{attribute 'linkalways'} 
{attribute 'no_explicit_call' := 'This FB is a CLASS and must be accessed using methods or properties'}
{attribute 'enable_dynamic_creation'}
FUNCTION_BLOCK _ETcVnRotationAngle EXTENDS EnumDatatypeBase
VAR
	localData : ETcVnRotationAngle;
	activeData : REFERENCE TO ETcVnRotationAngle;
	enumBaseDatatype : _DINT(localData);
END_VAR

METHOD PRIVATE AddLocalEnumeration
VAR_INPUT
	Enumeration : T_MAXSTRING;
	Value : ETcVnRotationAngle;
END_VAR
AddEnumeration(Enumeration, Value);
END_METHOD

PROPERTY PUBLIC Address : PVOID
GET
Address := ADR(activeData);
END_GET
END_PROPERTY

METHOD PUBLIC ClearReference
VAR_INPUT
END_VAR
activeData REF= localData;
SetBaseDatatypeReference();
END_METHOD

METHOD PUBLIC Clone : I_Datatype
VAR
    pClone : POINTER TO _ETcVnRotationAngle;
END_VAR
pClone := __NEW(_ETcVnRotationAngle(InitialValue := Value));
Clone := pClone^;
END_METHOD

METHOD FB_init : BOOL
VAR_INPUT
	bInitRetains : BOOL; // if TRUE, the retain variables are initialized (warm start / cold start)
	bInCopyCode : BOOL;  // if TRUE, the instance afterwards gets moved into the copy code (online change)
	InitialValue : ETcVnRotationAngle;
END_VAR
localData := InitialValue;
AddBaseDatatype(enumBaseDatatype);
ClearReference();

AddLocalEnumeration('TCVN_RA_90_DEG', ETcVnRotationAngle.TCVN_RA_90_DEG);
AddLocalEnumeration('TCVN_RA_180_DEG', ETcVnRotationAngle.TCVN_RA_180_DEG);
AddLocalEnumeration('TCVN_RA_270_DEG', ETcVnRotationAngle.TCVN_RA_270_DEG);
END_METHOD

PROPERTY PUBLIC Identifier : T_MAXSTRING
GET
Identifier := 'ETcVnRotationAngle';
END_GET
END_PROPERTY

METHOD IsEnumeratorValueEqual : BOOL
VAR_INPUT
	Enumerator : I_KeyValueForwardEnumerator;
END_VAR
VAR
	storedValue : ETcVnRotationAngle;
END_VAR
IF NOT Enumerator.TryGet(storedValue) THEN
	RETURN;
END_IF

IsEnumeratorValueEqual := storedValue = activeData;
END_METHOD

METHOD PUBLIC MakeReferenceTo
VAR_INPUT
	ReferenceTarget : REFERENCE TO ETcVnRotationAngle;
END_VAR
activeData REF= ReferenceTarget;
SetBaseDatatypeReference();
END_METHOD

METHOD PROTECTED SetBaseDatatypeReference
VAR_INPUT
END_VAR
enumBaseDatatype.MakeReferenceTo(activeData);
END_METHOD

PROPERTY PUBLIC Size : UDINT
GET
Size := SIZEOF(activeData);
END_GET
END_PROPERTY

METHOD TryMakeReferenceTo : BOOL
VAR_INPUT
	Target : I_Datatype;
END_VAR
VAR
	targetAsEnum : I_EnumDatatype;
	pTargetData : POINTER TO ETcVnRotationAngle;
END_VAR
IF NOT Target.TryResolveAsEnumDatatype(targetAsEnum) THEN
	RETURN;
END_IF

IF targetAsEnum.Identifier <> Identifier THEN
	RETURN;
END_IF

pTargetData := Target.Address;
activeData REF= pTargetData^;
SetBaseDatatypeReference();
TryMakeReferenceTo := TRUE;
END_METHOD

PROPERTY PUBLIC Value : ETcVnRotationAngle
GET
Value := activeData;
END_GET
SET
activeData := Value;
END_SET
END_PROPERTY

END_FUNCTION_BLOCK

(* stored: Version 1.1.0.1
   POU _ETcVnRotationAngle: Id {85d60ac7-044d-46f0-8359-758b7ec39bdd}, SpecialFunc None
   Folder Constructor: Id {e2ec5270-5f60-4294-8a6f-783e17a82fff}
   Folder Private: Id {1819f076-a18c-4767-ae39-639cdee8e07c}
   Folder Protected: Id {5a16ea8f-0523-4d3b-ad90-cc5985734c25}
   Method AddLocalEnumeration: Id {59b88426-96c5-4b22-be20-8f51fbede1d1}
   Property Address: Id {fbdcf1c1-bfe6-4feb-a638-9d5dbf03b40f}
   Get Get: Id {d1127421-6293-4aab-affc-3ccab4407517}
   Method ClearReference: Id {2819fe97-e805-4d3f-85be-09ddae06c1ad}
   Method Clone: Id {b3df2c52-3693-4d44-99b2-dd1f3328a048}
   Method FB_init: Id {de0923ab-8a9c-4b3b-9aea-99f2d4a54283}
   Property Identifier: Id {6c4eb71b-ffa9-4fce-8495-020ccc503055}
   Get Get: Id {e9cc94cc-b3ec-40c2-b89e-f4dbaaaa6a8b}
   Method IsEnumeratorValueEqual: Id {56e16fe7-9521-4a2c-a80f-1024c596b403}
   Method MakeReferenceTo: Id {9470b849-d89c-4969-84a3-e11d8229eb73}
   Method SetBaseDatatypeReference: Id {261ee742-adcd-47b1-9f24-f3b44c27e677}
   Property Size: Id {6d164746-73c6-4e08-9c6d-4075057dc0f4}
   Get Get: Id {c18dc6de-8046-4751-b069-20073daf418b}
   Method TryMakeReferenceTo: Id {927f8735-efa3-49d6-a10c-ab41953cd5cf}
   Property Value: Id {69398db9-489f-4d2e-9731-e0dc4114a01d}
   Get Get: Id {778b0732-1ba0-4243-b94e-acfafe2006bb}
   Set Set: Id {20464472-a383-4a32-94a9-960351d30a5b} *)
